(* CODESYS project test.project

Project tree, tasks and I/O mapping:
  CODESYS_Control_Win_V3 : CODESYS Control Win V3 x64, 3S - Smart Software Solutions GmbH, version 3.5.13.20
    application Application
      libraries: Standard, * (System); Time and Date, 3.5.7.0 (3S - Smart Software Solutions GmbH); BASIC, 3.3.3.0 (OSCAT); Memory, 3.5.7.0 (3S - Smart Software Solutions GmbH); Network, 3.5.7.0 (3S - Smart Software Solutions GmbH)
      task main (cyclic, interval t#20ms, priority 0) calls testNV
      global variables NetworkList
      global variables GlobalList
      program testNV [ST]
  function block FB1 [ST]
  text list GlobalTextList
*)

// CODESYS_Control_Win_V3/Application/NetworkList
VAR_GLOBAL
	// номер поста
	postNumber: INT;
	
	// Состояние терминала: ожидание, функции, окончание мойки, уборка, инкассация, пополнение баланса оператором
	postMode: INT;
	// TYPE EnumMode :
	// (
	// 	FUNC		:= 0,	// терминал готов к включению функций
	// 	
	// 	ACTIVECLEAN	:= 1,	// Р1. ECO-power		2
	// 	FOAM		:= 2,	// Р2. Пена				4
	// 	SHAMPOO		:= 3,	// Р3. Шампунь			3
	// 	COLDWATER	:= 4,	// Р4. Холодная вода	1
	// 	HOTWATER	:= 5,	// Р5. Горячая вода		2
	// 	WAX			:= 6,	// Р6. Воск				4
	// 	OSMOSE		:= 7,	// Р7. Осмос			3
	// 	PAUSE		:= 8,	// Пауза				4
	// 	
	// 	IDLE		:= 9,	// терминал в ожидании клиентов
	// 	ADVERT		:= 10,	// реклама	
	// 	
	// 	FIN			:= 500,	// Экран окончания мойки
	// 	CLEANUP		:= 600,	// Экран уборки
	// 	CASHCOLLECT	:= 700,	// Экран инкассации
	// 	CASHCOLLECT_FIN	:= 710,	// Экран окончания инкассации
	// 	FREEMONEY	:= 800	// Экран добавления денег
	// 	STOP		:= 1000	// Экран состояния останова поста
	// );
	// END_TYPE

	// баланс
	postCounterFund: INT;

	// тип карты
	cardType: INT;
	// TYPE EnumCardType :
	// (
	// 	UNDEFINED	:= 0,	// неопределённая карта (карта отсутствует)
	// 	CLEANUP		:= 1,	// карта уборки
	// 	CASHCOLLECT	:= 2,	// карта инкассации
	// 	FREEMONEY	:= 3,	// карта добавления денег (бесплатной мойки)
	// 	SERVICE		:= 4	// карта техслужбы
	// );
	// END_TYPE	

	
	// нажатая кнопка
	buttonActive: INT;
	// TYPE EnumButton :
	// (
	// 	NONE := 0,				// нет нажатой кнопки
	// 	BTN_ACTIVECLEAN := 1,	// Р1. ECO-power
	// 	BTN_FOAM := 2,			// Р2. Пена
	// 	BTN_SHAMPOO := 3,		// Р3. Шампунь
	// 	BTN_COLDWATER := 4,		// Р4. Холодная вода
	// 	BTN_HOTWATER := 5,		// Р5. Горячая вода
	// 	BTN_WAX := 6,			// Р6. Воск
	// 	BTN_OSMOSE := 7,		// Р7. Осмос
	// 	BTN_PAUSE := 8,			// Пауза
	// 	BTN_PRINT := 9,			// Печать чека
	// 	BTN_HELP := 10			// Вызов оператора
	// );
	// END_TYPE
		
	// сумма внесения
	amountReceived: INT;
	
	
	// стоимость оконченной мойки
	costWash: INT;
	// сдача
	costChange: INT;
	// стоимость активной химии
	costActiveClean: INT;
	// стоимость пены
	costFoam: INT;
	// стоимость шампуня
	costShampoo: INT;
	// стоимость ХВ
	costColdWater: INT;
	// стоимость ГВ
	costHotWater: INT;
	// стоимость воска
	costWax: INT;
	// стоимость осмоса
	costOsmose: INT;
	// стоимость паузы
	costPause: INT;

	
	// состояние верхнего замка
	lockTop: INT;
	// состояние среднего замка
	lockMid: INT;
	// 1 - замок закрыт; 0 - замок открыт
END_VAR

// CODESYS_Control_Win_V3/Application/GlobalList
{attribute 'qualified_only'}
VAR_GLOBAL
	
END_VAR

// CODESYS_Control_Win_V3/Application/testNV
PROGRAM testNV
VAR CONSTANT
	MODES_SIZE : BYTE := 11;
	
	//EJECT_TICKET_COMMAND : ARRAY[0..MODES_SIZE-1] OF INT := [0, 1, 2, 3 , 4 ,5,  6, 7, 8, 9, 10, 500, 600, 700, 710, 800, 1000];
	                // 	NONE := 0,				// нет нажатой кнопки
                // 	BTN_ACTIVECLEAN := 1,	// Р1. ECO-power
                // 	BTN_FOAM := 2,			// Р2. Пена
                // 	BTN_SHAMPOO := 3,		// Р3. Шампунь
                // 	BTN_COLDWATER := 4,		// Р4. Холодная вода
                // 	BTN_HOTWATER := 5,		// Р5. Горячая вода
                // 	BTN_WAX := 6,			// Р6. Воск
                // 	BTN_OSMOSE := 7,		// Р7. Осмос
                // 	BTN_PAUSE := 8,			// Пауза
                // 	BTN_PRINT := 9,			// Печать чека
                // 	BTN_HELP := 10			// Вызов оператора
	
	
	BUTTONS_MODES : ARRAY[0..MODES_SIZE-1] OF INT := [0, 1, 2, 3 , 4 ,5,  6, 7, 8, 9, 10];
END_VAR

VAR
	timer : TON;
	modeIndex : BYTE:=0;
	
	
	tSysStartTime		: TIME;
	dateAndTime : DATE_AND_TIME;
	
	currTime : UDINT;
	aux1 : UINT;
	aux2 : UINT;
END_VAR

IF timer.IN  THEN
	timer(IN:= TRUE);
	IF NOT (timer.Q) THEN
		RETURN;
	ELSE
		timer(IN:=FALSE);	
	END_IF
END_IF

                // 	FUNC		:= 0,	// терминал готов к включению функций
                //
                // 	ACTIVECLEAN	:= 1,	// Р1. ECO-power		2
                // 	FOAM		:= 2,	// Р2. Пена				4
                // 	SHAMPOO		:= 3,	// Р3. Шампунь			3
                // 	COLDWATER	:= 4,	// Р4. Холодная вода	1
                // 	HOTWATER	:= 5,	// Р5. Горячая вода		2
                // 	WAX			:= 6,	// Р6. Воск				4
                // 	OSMOSE		:= 7,	// Р7. Осмос			3
                // 	PAUSE		:= 8,	// Пауза				4
                //
                // 	IDLE		:= 9,	// терминал в ожидании клиентов
                // 	ADVERT		:= 10,	// реклама
                //
                // 	FIN			:= 500,	// Экран окончания мойки
                // 	CLEANUP		:= 600,	// Экран уборки
                // 	CASHCOLLECT	:= 700,	// Экран инкассации
                // 	CASHCOLLECT_FIN	:= 710,	// Экран окончания инкассации
                // 	FREEMONEY	:= 800	// Экран добавления денег
                // 	STOP		:= 1000	// Экран состояния останова поста

postMode:=0; 

postCounterFund :=  postCounterFund + 50;



buttonActive := BUTTONS_MODES[modeIndex];

modeIndex := modeIndex + 1;

IF modeIndex = MODES_SIZE THEN
	modeIndex := 0;
END_IF

(* time in milliseconds since the last system start *)
tSysStartTime := TIME();

currTime := TIME_TO_UDINT(tSysStartTime);

aux1 := UDINT_TO_UINT(SHR(currTime,16));
aux2 := UDINT_TO_UINT(currTime AND 16#FFFF);

lockTop := UINT_TO_INT(aux1); 
lockMid :=  UINT_TO_INT(aux2); 


timer(IN:= TRUE, PT := T#3S);

END_PROGRAM

// FB1
FUNCTION_BLOCK FB1
VAR_INPUT
	in:INT;
END_VAR
VAR_OUTPUT
	out:INT;
END_VAR
VAR
	ivar:INT:=2;
END_VAR

out:=in+ivar;

END_FUNCTION_BLOCK
